PROGRAM Sequence
VAR
	Counter_1: CTU;
	temp: WORD;
	counter_PV: WORD;
	
	tempPosition, tempI:REAL;
	Position, Amper: INT;
	
	
	
	
	
END_VAR
VAR // added by the converter: edge detectors and wires of the graphical bodies
    _w1, _w2 : BOOL;
END_VAR

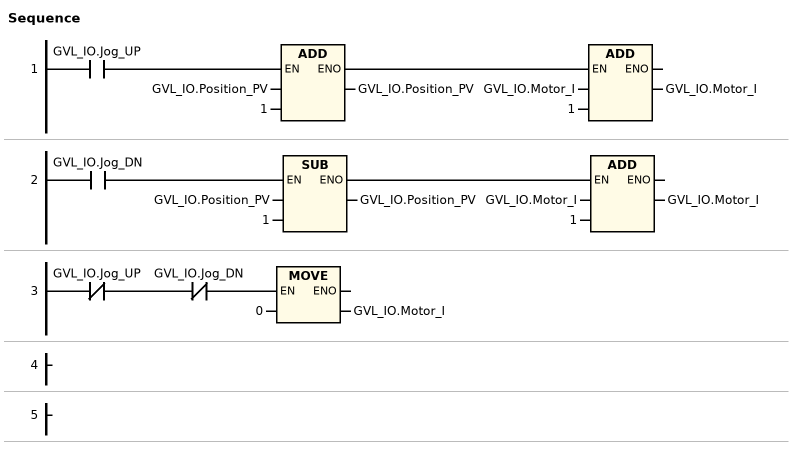
// NETWORK 1
_w1 := GVL_IO.Jog_UP;
IF _w1 THEN GVL_IO.Position_PV := GVL_IO.Position_PV + 1; END_IF
IF _w1 THEN GVL_IO.Motor_I := GVL_IO.Motor_I + 1; END_IF

// NETWORK 2
_w2 := GVL_IO.Jog_DN;
IF _w2 THEN GVL_IO.Position_PV := GVL_IO.Position_PV - 1; END_IF
IF _w2 THEN GVL_IO.Motor_I := GVL_IO.Motor_I + 1; END_IF

// NETWORK 3
IF NOT GVL_IO.Jog_UP AND NOT GVL_IO.Jog_DN THEN GVL_IO.Motor_I := 0; END_IF

// NETWORK 4

// NETWORK 5

END_PROGRAM

(* stored: Version 1.1.0.1, ProductVersion 3.1.4024.13
   POU Sequence: Id {c1e8b212-cdaa-4924-8e34-e8eac1ed4385}, SpecialFunc None *)
